(* CoDeSys 2.3.9.59 project: PD5.pro *)
(* Libraries: Standard.lib, SYSLIBCALLBACK.LIB *)

(* PLC configuration (modules and I/O channels)
Configuration EC4P-200 [Root] node -1, in %IB0 out %QB0 {EC4P_RestartPwrOn = WARMSTART; EC4P_MaxCycleTime = 20; EC4P_Com1BaudRate = 38400; EC4P_CAN1BaudRate = 125KBaud; EC4P_RoutingId = 127; EC4P_EasyNetId = 1; EC4P_EasyNetCfg = 0; EC4P_EasyNetCycleTime = 50; EC4P_RoutingChannel = CAN1; EC4P_IPFlags = 0; EC4P_IPAddress = 0; EC4P_SubNetMask = 0; EC4P_DefaultGateway = 0; EC4P_SummerWinterFlags = 0; EC4P_SummerWinterRule1 = 0; EC4P_SummerWinterRule2 = 0}
  Local I/O [EC4P_LocalIO] node 0, in %IB0 out %QB0 {EC4P_LocalInt = 0}
    I1 AT %IX0.0 [LocalBitInput] Input I1
    I2 AT %IX0.1 [LocalBitInput] Input I2
    I3 AT %IX0.2 [LocalBitInput] Input I3
    I4 AT %IX0.3 [LocalBitInput] Input I4
    I5 AT %IX0.4 [LocalBitInput] Input I5
    I6 AT %IX0.5 [LocalBitInput] Input I6
    I7 AT %IX0.6 [LocalBitInput] Input I7
    I8 AT %IX0.7 [LocalBitInput] Input I8
    I9 AT %IX1.0 [LocalBitInput] Input I9
    I10 AT %IX1.1 [LocalBitInput] Input I10
    I11 AT %IX1.2 [LocalBitInput] Input I11
    I12 AT %IX1.3 [LocalBitInput] Input I12
    I13 AT %IX1.4 [LocalDiagInput] Diagnostic Input I13
    I14 AT %IX1.5 [LocalDiagInput] Diagnostic Input I14
    I15 AT %IX1.6 [LocalDiagInput] Diagnostic Input I15
    I16 AT %IX1.7 [LocalDiagInput] Diagnostic Input I16
    I7_Analog AT %IW2 [LocalAnalogIn] Input I7, 10Bit, 0-10VDC
    I8_Analog AT %IW4 [LocalAnalogIn] Input I8, 10Bit, 0-10VDC
    I11_Analog AT %IW6 [LocalAnalogIn] Input I11, 10Bit, 0-10VDC
    I12_Analog AT %IW8 [LocalAnalogIn] Input I12, 10Bit, 0-10VDC
    Transistor Outputs [EC4P_TOutputs] node 0, in %IB10 out %QB0
      Q1 AT %QX0.0 [LocalBitOutput] Transistor-Output Q1
      Q2 AT %QX0.1 [LocalBitOutput] Transistor-Output Q2
      Q3 AT %QX0.2 [LocalBitOutput] Transistor-Output Q3
      Q4 AT %QX0.3 [LocalBitOutput] Transistor-Output Q4
      Q5 AT %QX0.4 [LocalBitOutput] Transistor-Output Q5
      Q6 AT %QX0.5 [LocalBitOutput] Transistor-Output Q6
      Q7 AT %QX0.6 [LocalBitOutput] Transistor-Output Q7
      Q8 AT %QX0.7 [LocalBitOutput] Transistor-Output Q8
    No Analog Output [EC4P_NoAnalogOutput] node 1, in %IB10 out %QB1
    No Keys [EC4P_NoKeys] node 2, in %IB10 out %QB1
    No Counter [EC4P_NoCounter] node 3, in %IB10 out %QB1
  Extension [EC4P_Extension] node 1, in %IB10 out %QB1
    No Extension [EC4P_NoExtension] node 0, in %IB10 out %QB1
*)

(* POU PLC_PRG, SFC *)
PROGRAM PLC_PRG
VAR
	init_done: BOOL;
	slider_value: INT;
	mode: WORD;
	state: WORD;
	bottom_val, top_val: INT;

	CTU: CTU;
	ctu_reset: BOOL;
	ctud_mode: CTUD;
	ctud_reset: BOOL;

	segment: segment_driver;
	sumator: input_sum;
	trigger_fall: F_TRIG;
	timer: TON;
	reset: BOOL;

	done: BOOL;
	done_b: BOOL;
	done_t: BOOL;

	gui_mode0: BOOL;
	gui_mode1: BOOL;
	gui_mode2: BOOL;
END_VAR
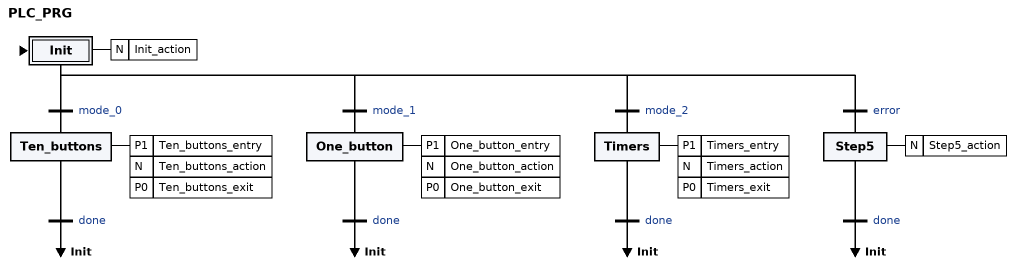
INITIAL_STEP Init:
	Init_action(N);
END_STEP
TRANSITION FROM Init TO Ten_buttons := mode_0;
END_TRANSITION
TRANSITION FROM Init TO One_button := mode_1;
END_TRANSITION
TRANSITION FROM Init TO Timers := mode_2;
END_TRANSITION
TRANSITION FROM Init TO Step5 := error;
END_TRANSITION
STEP Ten_buttons:
	Ten_buttons_entry(P1);
	Ten_buttons_action(N);
	Ten_buttons_exit(P0);
END_STEP
TRANSITION FROM Ten_buttons TO Init := done;
END_TRANSITION
STEP One_button:
	One_button_entry(P1);
	One_button_action(N);
	One_button_exit(P0);
END_STEP
TRANSITION FROM One_button TO Init := done;
END_TRANSITION
STEP Timers:
	Timers_entry(P1);
	Timers_action(N);
	Timers_exit(P0);
END_STEP
TRANSITION FROM Timers TO Init := done;
END_TRANSITION
STEP Step5:
	Step5_action(N);
END_STEP
TRANSITION FROM Step5 TO Init := done;
END_TRANSITION

ACTION Init_action:
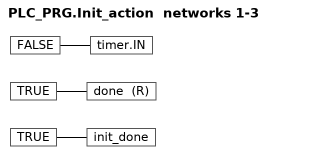
_FBD_ (* Function Block Diagram *)
NETWORK 1
	FALSE => timer.IN
NETWORK 2
	TRUE => R done
NETWORK 3
	TRUE => init_done
_END_FBD_
(* the same logic as Structured Text *)
(* Network 1 *)
timer.IN := FALSE;
(* Network 2 *)
done := FALSE;
(* Network 3 *)
init_done := TRUE;
END_ACTION

ACTION Ten_buttons_entry:
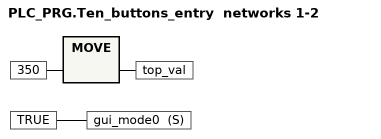
_FBD_ (* Function Block Diagram *)
NETWORK 1
	MOVE(350) => top_val
NETWORK 2
	TRUE => S gui_mode0
_END_FBD_
(* the same logic as Structured Text *)
(* Network 1 *)
top_val := 350;
(* Network 2 *)
gui_mode0 := TRUE;
END_ACTION

ACTION Ten_buttons_action:
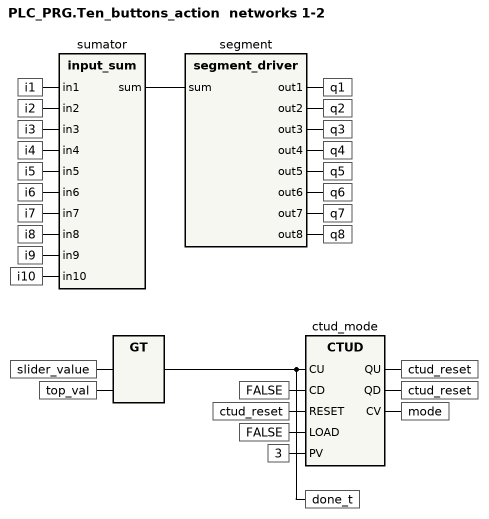
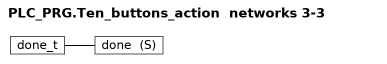
_FBD_ (* Function Block Diagram *)
NETWORK 1
	segment:segment_driver(sum: sumator:input_sum(in1: i1, in2: i2, in3: i3, in4: i4, in5: i5, in6: i6, in7: i7, in8: i8, in9: i9, in10: i10), out2 => q2, out3 => q3, out4 => q4, out5 => q5, out6 => q6, out7 => q7, out8 => q8) => q1
NETWORK 2
	ctud_mode:CTUD(CU: <GT(slider_value, top_val) => done_t>, CD: FALSE, RESET: ctud_reset, LOAD: FALSE, PV: 3, QD => ctud_reset, CV => mode) => ctud_reset
NETWORK 3
	done_t => S done
_END_FBD_
(* the same logic as Structured Text *)
(* Network 1 *)
sumator(in1 := i1, in2 := i2, in3 := i3, in4 := i4, in5 := i5, in6 := i6, in7 := i7, in8 := i8, in9 := i9, in10 := i10);
segment(sum := sumator.sum);
q2 := segment.out2;
q3 := segment.out3;
q4 := segment.out4;
q5 := segment.out5;
q6 := segment.out6;
q7 := segment.out7;
q8 := segment.out8;
q1 := segment.out1;
(* Network 2: see the listing above *)
(* Network 3 *)
IF done_t THEN done := TRUE; END_IF;
END_ACTION

ACTION Ten_buttons_exit:
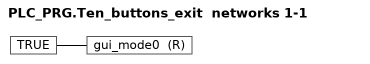
_FBD_ (* Function Block Diagram *)
NETWORK 1
	TRUE => R gui_mode0
_END_FBD_
(* the same logic as Structured Text *)
(* Network 1 *)
gui_mode0 := FALSE;
END_ACTION

ACTION One_button_entry:
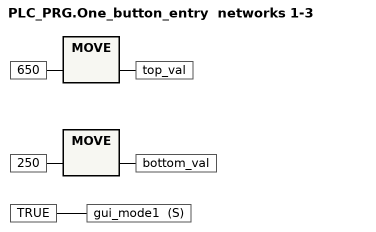
_FBD_ (* Function Block Diagram *)
NETWORK 1
	MOVE(650) => top_val
NETWORK 2
	MOVE(250) => bottom_val
NETWORK 3
	TRUE => S gui_mode1
_END_FBD_
(* the same logic as Structured Text *)
(* Network 1 *)
top_val := 650;
(* Network 2 *)
bottom_val := 250;
(* Network 3 *)
gui_mode1 := TRUE;
END_ACTION

ACTION One_button_action:
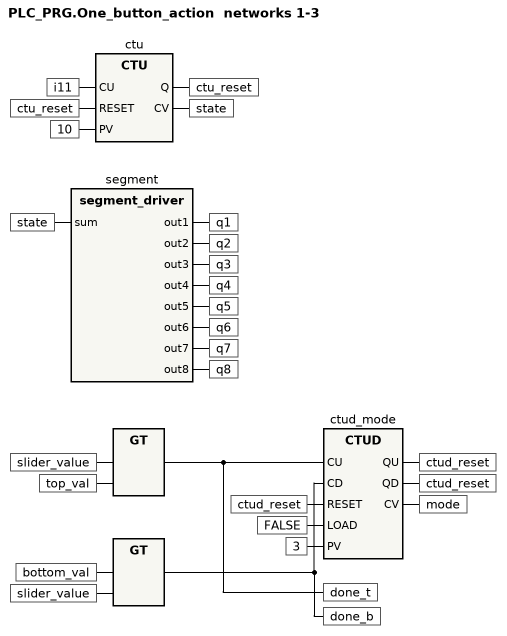
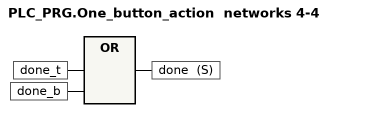
_FBD_ (* Function Block Diagram *)
NETWORK 1
	ctu:CTU(CU: i11, RESET: ctu_reset, PV: 10, CV => state) => ctu_reset
NETWORK 2
	segment:segment_driver(sum: state, out2 => q2, out3 => q3, out4 => q4, out5 => q5, out6 => q6, out7 => q7, out8 => q8) => q1
NETWORK 3
	ctud_mode:CTUD(CU: <GT(slider_value, top_val) => done_t>, CD: <GT(bottom_val, slider_value) => done_b>, RESET: ctud_reset, LOAD: FALSE, PV: 3, QD => ctud_reset, CV => mode) => ctud_reset
NETWORK 4
	OR(done_t, done_b) => S done
_END_FBD_
(* the same logic as Structured Text *)
(* Network 1 *)
ctu(CU := i11, RESET := ctu_reset, PV := 10);
state := ctu.CV;
ctu_reset := ctu.Q;
(* Network 2 *)
segment(sum := state);
q2 := segment.out2;
q3 := segment.out3;
q4 := segment.out4;
q5 := segment.out5;
q6 := segment.out6;
q7 := segment.out7;
q8 := segment.out8;
q1 := segment.out1;
(* Network 3: see the listing above *)
(* Network 4 *)
IF done_t OR done_b THEN done := TRUE; END_IF;
END_ACTION

ACTION One_button_exit:
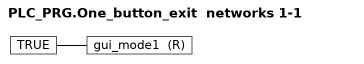
_FBD_ (* Function Block Diagram *)
NETWORK 1
	TRUE => R gui_mode1
_END_FBD_
(* the same logic as Structured Text *)
(* Network 1 *)
gui_mode1 := FALSE;
END_ACTION

ACTION Timers_entry:
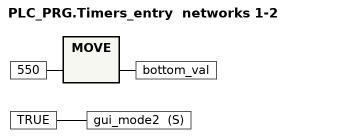
_FBD_ (* Function Block Diagram *)
NETWORK 1
	MOVE(550) => bottom_val
NETWORK 2
	TRUE => S gui_mode2
_END_FBD_
(* the same logic as Structured Text *)
(* Network 1 *)
bottom_val := 550;
(* Network 2 *)
gui_mode2 := TRUE;
END_ACTION

ACTION Timers_action:
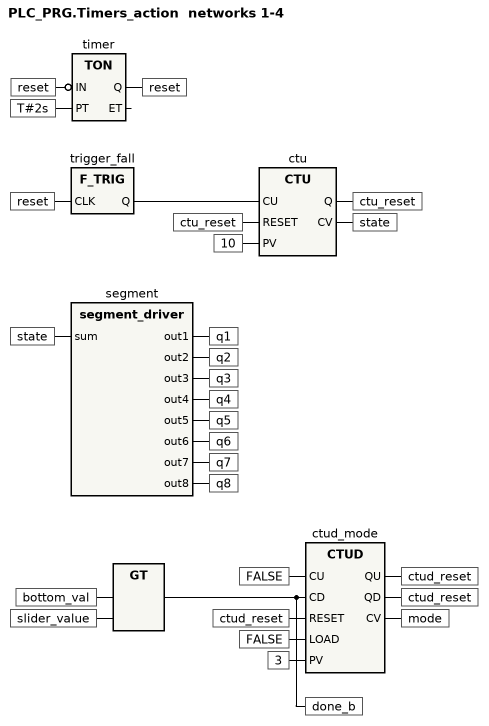
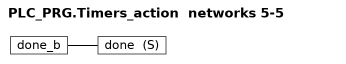
_FBD_ (* Function Block Diagram *)
NETWORK 1
	timer:TON(IN: NOT reset, PT: T#2s) => reset
NETWORK 2
	ctu:CTU(CU: trigger_fall:F_TRIG(CLK: reset), RESET: ctu_reset, PV: 10, CV => state) => ctu_reset
NETWORK 3
	segment:segment_driver(sum: state, out2 => q2, out3 => q3, out4 => q4, out5 => q5, out6 => q6, out7 => q7, out8 => q8) => q1
NETWORK 4
	ctud_mode:CTUD(CU: FALSE, CD: <GT(bottom_val, slider_value) => done_b>, RESET: ctud_reset, LOAD: FALSE, PV: 3, QD => ctud_reset, CV => mode) => ctud_reset
NETWORK 5
	done_b => S done
_END_FBD_
(* the same logic as Structured Text *)
(* Network 1 *)
timer(IN := NOT reset, PT := T#2s);
reset := timer.Q;
(* Network 2 *)
trigger_fall(CLK := reset);
ctu(CU := trigger_fall.Q, RESET := ctu_reset, PV := 10);
state := ctu.CV;
ctu_reset := ctu.Q;
(* Network 3 *)
segment(sum := state);
q2 := segment.out2;
q3 := segment.out3;
q4 := segment.out4;
q5 := segment.out5;
q6 := segment.out6;
q7 := segment.out7;
q8 := segment.out8;
q1 := segment.out1;
(* Network 4: see the listing above *)
(* Network 5 *)
IF done_b THEN done := TRUE; END_IF;
END_ACTION

ACTION Timers_exit:
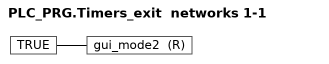
_FBD_ (* Function Block Diagram *)
NETWORK 1
	TRUE => R gui_mode2
_END_FBD_
(* the same logic as Structured Text *)
(* Network 1 *)
gui_mode2 := FALSE;
END_ACTION

ACTION Step5_action:
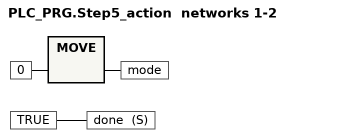
_FBD_ (* Function Block Diagram *)
NETWORK 1
	MOVE(0) => mode
NETWORK 2
	TRUE => S done
_END_FBD_
(* the same logic as Structured Text *)
(* Network 1 *)
mode := 0;
(* Network 2 *)
done := TRUE;
END_ACTION

TRANSITION mode_0:
_FBD_ (* Function Block Diagram *)
NETWORK 1
	AND(EQ(mode, 0), init_done)
_END_FBD_
END_TRANSITION

TRANSITION mode_1:
_FBD_ (* Function Block Diagram *)
NETWORK 1
	AND(EQ(mode, 1), init_done)
_END_FBD_
END_TRANSITION

TRANSITION mode_2:
_FBD_ (* Function Block Diagram *)
NETWORK 1
	AND(EQ(mode, 2), init_done)
_END_FBD_
END_TRANSITION

TRANSITION error:
_FBD_ (* Function Block Diagram *)
NETWORK 1
	AND(GT(mode, 2), init_done)
_END_FBD_
END_TRANSITION
END_PROGRAM

(* POU segment_driver, ST *)
FUNCTION_BLOCK segment_driver
VAR_INPUT
	sum: WORD;
END_VAR
VAR_OUTPUT
	out1, out2, out3, out4, out5, out6, out7, out8: BOOL;
END_VAR
VAR
END_VAR
CASE sum OF
0:
	out1 := 0;
	out2 := 0;
	out3 := 0;
	out4 := 0;
	out5 := 0;
	out6 := 0;
	out7 := 0;
	out8 := 1;
1:
	out1 := 0;
	out2 := 1;
	out3 := 0;
	out4 := 1;
	out5 := 1;
	out6 := 1;
	out7 := 1;
	out8 := 0;
2:
	out1 := 0;
	out2 := 0;
	out3 := 0;
	out4 := 1;
	out5 := 1;
	out6 := 0;
	out7 := 0;
	out8 := 0;
3:
	out1 := 1 ;
	out2 := 0;
	out3 := 1;
	out4 := 1;
	out5 := 1;
	out6 := 0;
	out7 := 1;
	out8 := 0;
4:
	out1 := 1;
	out2 := 1;
	out3 := 0;
	out4 := 1;
	out5 := 1;
	out6 := 0;
	out7 := 1;
	out8 := 0;
5:
	out1 := 1;
	out2 := 0;
	out3 := 1;
	out4 := 1;
	out5 := 1;
	out6 := 0;
	out7 := 1;
	out8 := 0;
6:
	out1 := 0;
	out2 := 1;
	out3 := 0;
	out4 := 0;
	out5 := 1;
	out6 := 0;
	out7 := 0;
	out8 := 0;
7:
	out1 := 0;
	out2 := 0;
	out3 := 0;
	out4 := 1;
	out5 := 1;
	out6 := 1;
	out7 := 0;
	out8 := 0;
8:
	out1 := 1;
	out2 := 1;
	out3 := 0;
	out4 := 1;
	out5 := 0;
	out6 := 1;
	out7 := 1;
	out8 := 0;
9:
	out1 := 1;
	out2 := 1;
	out3 := 0;
	out4 := 1;
	out5 := 1;
	out6 := 1;
	out7 := 0;
	out8 := 0;
10:
	out1 := 1;
	out2 := 1;
	out3 := 1;
	out4 := 1;
	out5 := 1;
	out6 := 1;
	out7 := 0;
	out8 := 0;
ELSE
	out1 := 0;
	out2 := 0;
	out3 := 0;
	out4 := 0;
	out5 := 0;
	out6 := 0;
	out7 := 0;
	out8 := 0;
END_CASE;
END_FUNCTION_BLOCK

(* POU input_sum, ST *)
FUNCTION_BLOCK input_sum
VAR_INPUT
	in1, in2, in3, in4, in5, in6, in7, in8, in9, in10: BOOL;
END_VAR
VAR_OUTPUT
	sum: WORD;
END_VAR
VAR
END_VAR
sum := BOOL_TO_INT(in1) + BOOL_TO_INT(in2) + BOOL_TO_INT(in3) + BOOL_TO_INT(in4) + BOOL_TO_INT(in5) + BOOL_TO_INT(in6)+ BOOL_TO_INT(in7) + BOOL_TO_INT(in8) + BOOL_TO_INT(in9) + BOOL_TO_INT(in10);
END_FUNCTION_BLOCK

(* Visualisation gui
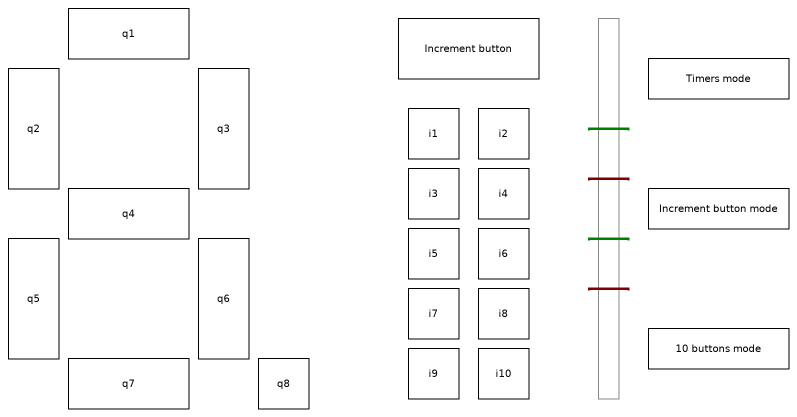
rectangle at (450,40)-(591,101): text "Increment button"; alarm colour if i11; taps i11
rectangle at (460,130)-(511,181): text "i1"; alarm colour if i1; toggles i1
rectangle at (530,130)-(581,181): text "i2"; alarm colour if i2; toggles i2
rectangle at (460,190)-(511,241): text "i3"; alarm colour if i3; toggles i3
rectangle at (530,190)-(581,241): text "i4"; alarm colour if i4; toggles i4
rectangle at (460,250)-(511,301): text "i5"; alarm colour if i5; toggles i5
rectangle at (460,310)-(511,361): text "i7"; alarm colour if i7; toggles i7
rectangle at (460,370)-(511,421): text "i9"; alarm colour if i9; toggles i9
rectangle at (530,250)-(581,301): text "i6"; alarm colour if i6; toggles i6
rectangle at (530,310)-(581,361): text "i8"; alarm colour if i8; toggles i8
rectangle at (530,370)-(581,421): text "i10"; alarm colour if i10; toggles i10
rectangle at (120,30)-(241,81): text "q1"; alarm colour if q1; toggles q1
rectangle at (250,90)-(301,211): text "q3"; alarm colour if q3; toggles q3
rectangle at (120,210)-(241,261): text "q4"; alarm colour if q4; toggles q4
rectangle at (60,90)-(111,211): text "q2"; alarm colour if q2; toggles q2
rectangle at (60,260)-(111,381): text "q5"; alarm colour if q5; toggles q5
rectangle at (250,260)-(301,381): text "q6"; alarm colour if q6; toggles q6
rectangle at (120,380)-(241,431): text "q7"; alarm colour if q7; toggles q7
rectangle at (310,380)-(361,431): text "q8"; alarm colour if q8; toggles q8
rectangle at (700,350)-(841,391): text "10 buttons mode"; alarm colour if PLC_PRG.gui_mode0; toggles PLC_PRG.gui_mode0
rectangle at (700,210)-(841,251): text "Increment button mode"; alarm colour if PLC_PRG.gui_mode1; toggles PLC_PRG.gui_mode1
rectangle at (700,80)-(841,121): text "Timers mode"; alarm colour if PLC_PRG.gui_mode2; toggles PLC_PRG.gui_mode2
rectangle at (640,260)-(681,261): invisible if NOT PLC_PRG.gui_mode0
rectangle at (640,310)-(681,311): invisible if NOT PLC_PRG.gui_mode1
rectangle at (640,150)-(681,151): invisible if NOT PLC_PRG.gui_mode1
rectangle at (640,200)-(681,201): invisible if NOT PLC_PRG.gui_mode2
1 more shapes without text or variables
*)
